// SIMATIC S7-200 SMART project (STEP 7-Micro/WIN SMART), CPU ST40

SYMBOL_TABLE 系统符号
Always_On        SM0.0    // 始终接通
Clock_1s         SM0.5    // 针对 1 s 的周期时间，时钟脉冲接通 0.5 s，断开 0.5 s.
END_SYMBOL_TABLE

ORGANIZATION_BLOCK MAIN:OB1
TITLE=程序注释
BEGIN
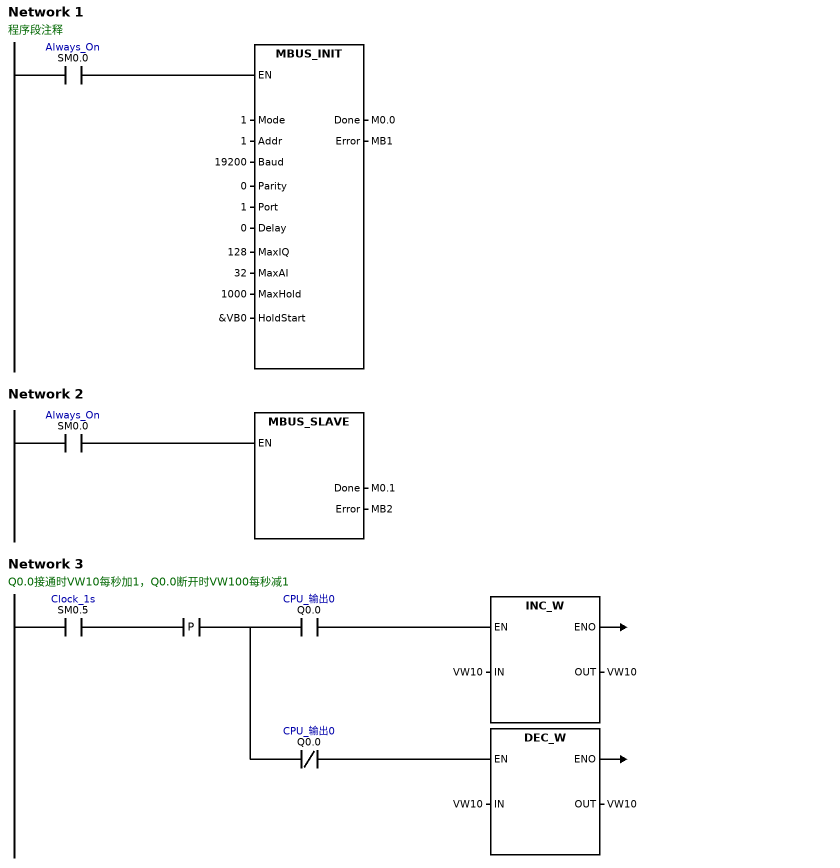
Network 1
// 程序段注释
LD     Always_On:SM0.0
CALL   MBUS_INIT:SBR1, 1, 1, 19200, 0, 1, 0, 128, 32, 1000, &VB0, M0.0, MB1
Network 2
LD     Always_On:SM0.0
CALL   MBUS_SLAVE:SBR2, M0.1, MB2
Network 3
// Q0.0接通时VW10每秒加1，Q0.0断开时VW100每秒减1
LD     Clock_1s:SM0.5
EU
LPS
A      CPU_输出0:Q0.0
INCW   VW10
LPP
AN     CPU_输出0:Q0.0
DECW   VW10
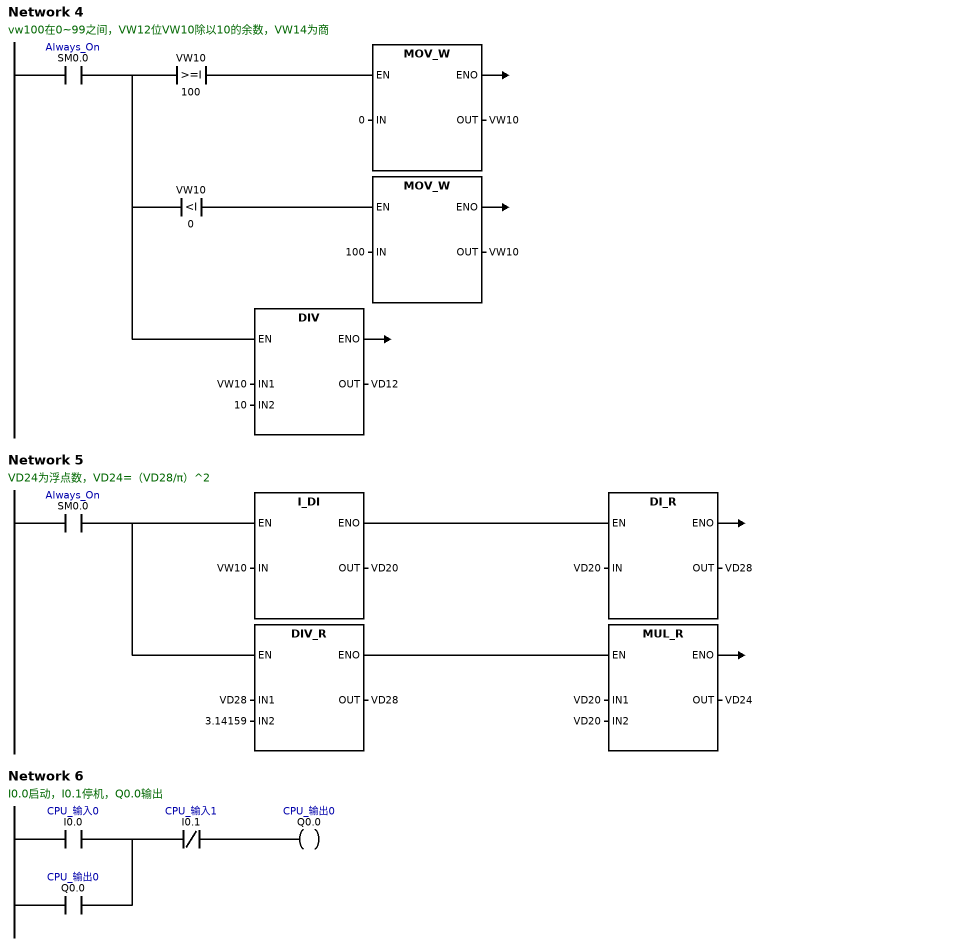
Network 4
// vw100在0~99之间，VW12位VW10除以10的余数，VW14为商
LD     Always_On:SM0.0
LPS
AW>=   VW10, 100
MOVW   0, VW10
LRD
AW<    VW10, 0
MOVW   100, VW10
LPP
MOVW   VW10, VW14
DIV    10, VD12
Network 5
// VD24为浮点数，VD24=（VD28/π）^2
LD     Always_On:SM0.0
LPS
ITD    VW10, VD20
AENO
DTR    VD20, VD28
LPP
/R     3.14159, VD28
AENO
MOVR   VD20, VD24
*R     VD20, VD24
Network 6
// I0.0启动，I0.1停机，Q0.0输出
LD     CPU_输入0:I0.0
O      CPU_输出0:Q0.0
AN     CPU_输入1:I0.1
=      CPU_输出0:Q0.0
END_ORGANIZATION_BLOCK

// SBR1: protected block, not included

// SBR2: protected block, not included

// SBR3: protected block, not included
